FUNCTION AssertEquals_STRING : BOOL
VAR_INPUT
    Source   : T_MaxString;
    Expected : T_MaxString;
    Actual   : T_MaxString;
    Message  : T_MaxString;
END_VAR
VAR_OUTPUT
    Failed : BOOL;
END_VAR

IF Expected <> Actual THEN
    F_LogResult(Source, FormatStringEx1('Assertion Failed - %s', Message));
    Failed := TRUE;
    RETURN;
END_IF

AssertEquals_STRING := TRUE;

END_FUNCTION

(* stored: Version 1.1.0.1, ProductVersion 3.1.4024.12
   POU AssertEquals_STRING: Id {3f350298-84b3-49fe-9a33-20a55bb8ec87}, SpecialFunc None *)
